Staubli VAL3: iHeater.pgx

public program iHeater(num& nNum[] (dimensions=1))
begin
  nNum=dioGet(iHeaterStatus)
end
